FUNCTION_BLOCK FB_SEL_WSTRING (* F_SEL replacement for WSTRING (F_SEL currently doesn't work with WSTRING) *)
  (* Standard: 61499-2 *)
  (* Version 1.0, 2017-08-27, Marc Jakobi, HTW Berlin *)
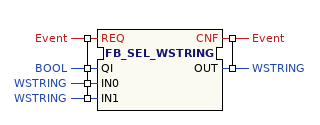
  EVENT_INPUT
    REQ WITH QI, IN0, IN1; (* Normal Execution Request *)
  END_EVENT
  EVENT_OUTPUT
    CNF WITH OUT; (* Execution Confirmation *)
  END_EVENT
  VAR_INPUT
    QI : BOOL; (* Input event qualifier *)
    IN0 : WSTRING; (* Selectable input variable *)
    IN1 : WSTRING; (* Selectable input variable *)
  END_VAR
  VAR_OUTPUT
    OUT : WSTRING; (* Selected output variable *)
  END_VAR
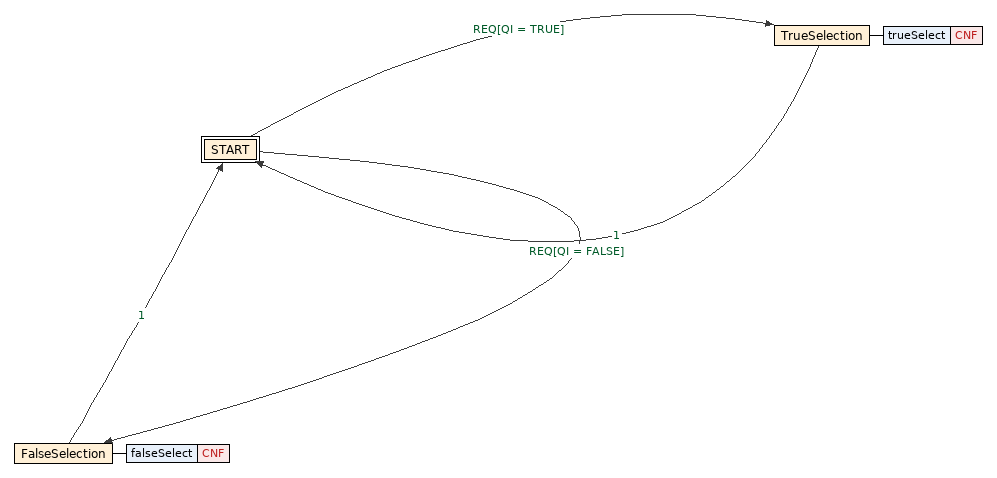
  EC_STATES
    START; (* Initial State *)
    TrueSelection : trueSelect -> CNF; (* Normal execution *)
    FalseSelection : falseSelect -> CNF;
  END_STATES
  EC_TRANSITIONS
    START TO TrueSelection := REQ[QI = TRUE];
    TrueSelection TO START := 1;
    START TO FalseSelection := REQ[QI = FALSE];
    FalseSelection TO START := 1;
  END_TRANSITIONS
  ALGORITHM trueSelect IN ST: (* called upon true input *)
OUT := IN1;
  END_ALGORITHM
  ALGORITHM falseSelect IN ST: (* called upon false input *)
OUT := IN0;
  END_ALGORITHM
END_FUNCTION_BLOCK
